FUNCTION_BLOCK "CIPSystem"
{ S7_Optimized_Access := 'TRUE' }
VERSION : 0.1
AUTHOR : 'AI_Generated'

VAR_INPUT
    bStart : Bool;                     // 启动清洗循环
    bStop : Bool;                      // 停止
    bReset : Bool;                     // 故障复位
    bEmergencyStop : Bool;             // 急停（常闭）
    bTankFull : Bool;                  // 清洗罐满
    bTankEmpty : Bool;                 // 清洗罐空
    bFlowOK : Bool;                    // 流量正常
    rTemperature : Real;               // 温度传感器 (degC)
    rConductivity : Real;              // 电导率 (uS/cm)
    bReturnFlowOK : Bool;              // 回流流量正常
END_VAR

VAR_OUTPUT
    bSupplyPump : Bool;                // 供液泵
    bReturnPump : Bool;                // 回流泵
    bHeater : Bool;                    // 加热器
    bRinseValve : Bool;                // 清水阀
    bCausticValve : Bool;              // 碱液阀
    bAcidValve : Bool;                 // 酸液阀
    bDrainValve : Bool;                // 排空阀
    bPhaseActive : Bool;               // 阶段运行中
    bCycleComplete : Bool;             // 循环完成
    bFault : Bool;                     // 故障
    iCurrentPhase : Int;               // 当前阶段
    iFaultCode : Int;                  // 故障代码
END_VAR

VAR_IN_OUT
    // 清洗参数（可从 DB 配置）
    tRinse1Time : Time;                // 第一次清水冲洗时间
    tCausticTime : Time;               // 碱洗时间
    tRinse2Time : Time;                // 第二次清水冲洗时间
    tAcidTime : Time;                  // 酸洗时间
    tFinalRinseTime : Time;            // 最终清水冲洗时间
    rCausticTempSetpoint : Real;       // 碱洗温度设定值 (degC)
    rAcidTempSetpoint : Real;          // 酸洗温度设定值 (degC)
    rRinseTempSetpoint : Real;         // 冲洗温度设定值 (degC)
    rCausticCondMin : Real;            // 碱液最小电导率 (uS/cm)
    rAcidCondMin : Real;               // 酸液最小电导率 (uS/cm)
    rRinseCondMax : Real;              // 冲洗最大电导率 (uS/cm)
END_VAR

VAR
    // 阶段常量
    c_IDLE : Int := 0;
    c_RINSE1 : Int := 1;
    c_CAUSTIC : Int := 2;
    c_RINSE2 : Int := 3;
    c_ACID : Int := 4;
    c_FINAL_RINSE : Int := 5;

    // 阶段计时器
    tPhaseTimer : TON;                 // 阶段计时
    tTempReach : TON;                  // 升温等待

    // 边沿检测
    bStartOld : Bool;
    bStartRising : Bool;

    // 阶段内状态
    bHeatingActive : Bool;             // 加热中
    bCondCheckPassed : Bool;           // 浓度检测通过
    bTempReached : Bool;               // 温度达到
    bRinseCondOK : Bool;               // 冲洗电导率达标

    // 停留监控
    tStallTimer : TON;                 // 阶段完成条件停留超时计时
    tStallTimeout : Time := T#30S;     // 停留超时时间
END_VAR

BEGIN
    // ── 急停 ──
    IF NOT bEmergencyStop THEN
        bSupplyPump := FALSE; bReturnPump := FALSE; bHeater := FALSE;
        bRinseValve := FALSE; bCausticValve := FALSE;
        bAcidValve := FALSE; bDrainValve := FALSE;
        bPhaseActive := FALSE; bFault := TRUE; iFaultCode := 1;
        iCurrentPhase := c_IDLE;
        tPhaseTimer(IN := FALSE);
        RETURN;
    END_IF;

    // ── 故障复位 ──
    IF bFault AND bReset THEN
        bFault := FALSE; iFaultCode := 0;
    END_IF;

    IF bFault THEN RETURN; END_IF;

    // ── 上升沿检测 ──
    bStartRising := bStart AND NOT bStartOld;
    bStartOld := bStart;

    // ── 停止 ──
    IF bStop AND iCurrentPhase <> c_IDLE THEN
        bSupplyPump := FALSE; bReturnPump := FALSE; bHeater := FALSE;
        bRinseValve := FALSE; bCausticValve := FALSE;
        bAcidValve := FALSE; bDrainValve := FALSE;
        bPhaseActive := FALSE; iCurrentPhase := c_IDLE;
        tPhaseTimer(IN := FALSE);
    END_IF;

    // ── 启动 ──
    IF bStartRising AND iCurrentPhase = c_IDLE THEN
        iCurrentPhase := c_RINSE1;
        bCycleComplete := FALSE;
    END_IF;

    // ── 安全联锁：罐满/罐空/回流丢失 → 立即停机（fail-closed）──
    IF iCurrentPhase <> c_IDLE AND NOT bDrainValve AND
       (bTankFull OR bTankEmpty OR NOT bReturnFlowOK) THEN
        bSupplyPump := FALSE; bReturnPump := FALSE; bHeater := FALSE;
        bRinseValve := FALSE; bCausticValve := FALSE;
        bAcidValve := FALSE; bDrainValve := FALSE;
        bPhaseActive := FALSE; bFault := TRUE; iFaultCode := 2;
        iCurrentPhase := c_IDLE;
        tPhaseTimer(IN := FALSE);
        RETURN;
    END_IF;

    // ── 清洗阶段执行 ──
    CASE iCurrentPhase OF

        1:  // RINSE1 — 第一次清水冲洗
            bSupplyPump := TRUE; bReturnPump := TRUE;
            bRinseValve := TRUE; bPhaseActive := TRUE;
            tPhaseTimer(IN := TRUE, PT := tRinse1Time);

            IF (tPhaseTimer.Q AND bFlowOK AND bReturnFlowOK) THEN
                bRinseValve := FALSE;
                bDrainValve := TRUE;
                tPhaseTimer(IN := FALSE);
                iCurrentPhase := c_CAUSTIC;
            END_IF;

        2:  // CAUSTIC — 碱洗循环
            bSupplyPump := TRUE; bReturnPump := TRUE;
            bCausticValve := TRUE; bDrainValve := FALSE; bPhaseActive := TRUE;

            // 升温控制
            IF rTemperature < rCausticTempSetpoint THEN
                bHeater := TRUE; bHeatingActive := TRUE;
            ELSE
                bHeater := FALSE; bHeatingActive := FALSE;
            END_IF;

            // 电导率检测：确认碱液浓度足够
            bCondCheckPassed := rConductivity >= rCausticCondMin;

            tPhaseTimer(IN := TRUE, PT := tCausticTime);
            IF tPhaseTimer.Q AND bCondCheckPassed AND bFlowOK AND bReturnFlowOK THEN
                bCausticValve := FALSE; bHeater := FALSE;
                bDrainValve := TRUE;
                tPhaseTimer(IN := FALSE);
                iCurrentPhase := c_RINSE2;
            END_IF;

        3:  // RINSE2 — 第二次清水冲洗
            bSupplyPump := TRUE; bReturnPump := TRUE;
            bRinseValve := TRUE; bDrainValve := FALSE; bPhaseActive := TRUE;
            tPhaseTimer(IN := TRUE, PT := tRinse2Time);

            IF (tPhaseTimer.Q AND bFlowOK AND bReturnFlowOK) THEN
                // 检查冲洗水电导率是否达标
                bRinseCondOK := rConductivity <= rRinseCondMax;
                IF bRinseCondOK THEN
                    bRinseValve := FALSE;
                    bDrainValve := TRUE;
                    tPhaseTimer(IN := FALSE);
                    iCurrentPhase := c_ACID;
                END_IF;
            END_IF;

        4:  // ACID — 酸洗循环
            bSupplyPump := TRUE; bReturnPump := TRUE;
            bAcidValve := TRUE; bDrainValve := FALSE; bPhaseActive := TRUE;

            // 升温控制
            IF rTemperature < rAcidTempSetpoint THEN
                bHeater := TRUE; bHeatingActive := TRUE;
            ELSE
                bHeater := FALSE; bHeatingActive := FALSE;
            END_IF;

            // 电导率检测：确认酸液浓度足够
            bCondCheckPassed := rConductivity >= rAcidCondMin;

            tPhaseTimer(IN := TRUE, PT := tAcidTime);
            IF tPhaseTimer.Q AND bCondCheckPassed AND bFlowOK AND bReturnFlowOK THEN
                bAcidValve := FALSE; bHeater := FALSE;
                bDrainValve := TRUE;
                tPhaseTimer(IN := FALSE);
                iCurrentPhase := c_FINAL_RINSE;
            END_IF;

        5:  // FINAL_RINSE — 最终清水冲洗
            bSupplyPump := TRUE; bReturnPump := TRUE;
            bRinseValve := TRUE; bDrainValve := FALSE; bPhaseActive := TRUE;
            tPhaseTimer(IN := TRUE, PT := tFinalRinseTime);

            bRinseCondOK := rConductivity <= rRinseCondMax;
            IF tPhaseTimer.Q AND bRinseCondOK AND bFlowOK AND bReturnFlowOK THEN
                bRinseValve := FALSE;
                bSupplyPump := FALSE; bReturnPump := FALSE;
                tPhaseTimer(IN := FALSE);
                bCycleComplete := TRUE;
                iCurrentPhase := c_IDLE;
            END_IF;

        0:  // IDLE
            bSupplyPump := FALSE; bReturnPump := FALSE; bHeater := FALSE;
            bRinseValve := FALSE; bCausticValve := FALSE;
            bAcidValve := FALSE; bDrainValve := FALSE;
            bPhaseActive := FALSE;

    END_CASE;

    // ── 停留超时：阶段计时到点但完成条件不满足 → fail-closed 停机 ──
    IF iCurrentPhase <> c_IDLE AND tPhaseTimer.Q THEN
        tStallTimer(IN := TRUE, PT := tStallTimeout);
        IF tStallTimer.Q THEN
            bFault := TRUE; iFaultCode := 3;
            bSupplyPump := FALSE; bReturnPump := FALSE; bHeater := FALSE;
            bRinseValve := FALSE; bCausticValve := FALSE;
            bAcidValve := FALSE; bDrainValve := FALSE;
            bPhaseActive := FALSE;
            tPhaseTimer(IN := FALSE);
            iCurrentPhase := c_IDLE;
        END_IF;
    ELSE
        tStallTimer(IN := FALSE);
    END_IF;

END_FUNCTION_BLOCK
